Fanuc KAREL source: kt00183.KL

-- PROVISIONAL review KL for V770-1; original PC SHA256 82f9342ec97e78eca979553fe982212d457d79a7df99885d228b4ee67784b612
-- Incomplete behavior may be omitted. Consult companion uncertainty JSON. Do not deploy.
PROGRAM KT00183
%NOLOCKGROUP
VAR
  OUT : INTEGER
-- UNRESOLVED_DECL Y1 type=002018
-- UNRESOLVED_DECL H2 type=002017
BEGIN
  -- UNRESOLVED_PC offsets 5-19; opcodes 2E,22,9D,33,B2
  -- UNRESOLVED_PC offsets 24-38; opcodes 2E,22,9D,33,B4
  -- UNRESOLVED_PC offsets 43-68; opcodes 22,9D,33,B1,22,9D,33,B3,56,23
  -- UNRESOLVED_PC offsets 73-77; opcodes 7F
END KT00183
